// TIA Portal V17 export
// export: Created 2025-08-05T09:36:01.7579286Z, ExportSetting WithDefaults, DisplayName Totally Integrated Automation Portal, DisplayVersion V17, DisplayName TIA Portal Openness, DisplayVersion V17, DisplayName TIA Portal Version Control Interface, DisplayVersion V17, DisplayName SINAMICS Startdrive Advanced, DisplayVersion V17, DisplayName SINAMICS Startdrive G130, G150, S120, S150, SINAMICS MV, S210, DisplayVersion V17, DisplayName SINAMICS Startdrive G110M, G120, G120C, G120D, G120P, G115D, DisplayVersion V17, DisplayName STEP 7 Professional, DisplayVersion V17, DisplayName STEP 7 Safety, DisplayVersion V17, DisplayName WinCC Advanced, DisplayVersion V17
TYPE "Scanner_Outputs"
// stored: IsFailsafeCompliant false
   STRUCT
      Start : Bool;   // Command to Start IPG Weld Job
      Enable : Bool;   // Enable Scanner (Always On)
      Control_Reserved : Bool;
      Control_Reserved_1 : Bool;
      Control_Reserved_2 : Bool;
      Control_Reserved_3 : Bool;
      Control_Reserved_4 : Bool;
      Control_Reserved_5 : Bool;
      Control_Reserved_6 { S7_SetPoint := 'True'} : Byte;
      Control_Reserved_7 : Int;
      "GPI_0/Strobe" : Bool;   // Strobe for IPG Weld to Load a New Job
      GPI_1 : Bool;
      GPI_2 : Bool;
      GPI_3 : Bool;
      GPI_4 : Bool;
      GPI_5 : Bool;
      GPI_6 : Bool;
      GPI_7 : Bool;
      GPI_8 : Bool;
      GPI_9 : Bool;
      GPI_10 : Bool;
      GPI_11 : Bool;
      GPI_12 : Bool;
      GPI_13 : Bool;
      GPI_14 : Bool;
      GPI_15 : Bool;
      Group_ID_Select : Byte;   // Group to be Loaded
      Job_ID_Select : Byte;   // Job to Be Loaded
      Register_A : DInt;
      Register_B : DInt;
      Register_C : DInt;
   END_STRUCT;
END_TYPE
